PROGRAM Socket
VAR
	fbFRSocket:fb_socket_FR;
	i:INT;
END_VAR


IF (g_maniTest.m_testStart[1]=TRUE) OR (g_maniTest.m_testStart[2]=TRUE) THEN
	fbFRSocket();
END_IF

// data monitor
FOR i:=1 TO 6 BY 1 DO
	g_maniTest.m_robotJntPos[i]:=fbFRSocket.datalreal[i-1];
	g_maniTest.m_sensorData[i]:=fbFRSocket.dataTorqueForce[i-1];		
END_FOR

END_PROGRAM

(* stored: Version 1.1.0.1, ProductVersion 3.1.4024.11
   POU Socket: Id {3ea1f794-102b-4ade-8899-710f8bdc81c0}, SpecialFunc None *)
